TYPE T_XV03_ValveSystem : 
	ARRAY[1..24] OF ST_XV03_ValveInfoData; 
END_TYPE

(* stored: Version 1.1.0.1, ProductVersion 3.1.4024.13
   DUT T_XV03_ValveSystem: Id {d28346da-3143-07dd-212e-868793821984} *)
